// TIA Portal project "FactoryIO_Template_S7-1200_V16_V16" (V16)
// Vorlageprojekt für das Buch mit Zielsystem S7-1200

(* hardware
DEVICE "S7-1200-Station_1"  S7-1200 Station
   slot 0: "Baugruppenträger_0"  Rack  V1.0
   slot 1: "PLC_1"  CPU 1211C DC/DC/DC  6ES7 211-1AE40-0XB0  V4.1
*)

// ===== PLC "PLC_1"  CPU 1211C DC/DC/DC =====

VAR_GLOBAL   // PLC tag table "Standard-Variablentabelle"
   "EMITTER(1)" AT %A0.0 : Bool;
   "START(1)" AT %E0.0 : Bool;
   "STOP(1)" AT %E0.1 : Bool;
   "ROLLER 1" AT %Q0.1 : Bool;
   "ROLLER 2" AT %Q0.2 : Bool;
   "B LIMIT" AT %I0.3 : Bool;
   "ROLLER 4" AT %Q0.3 : Bool;
   "LIMIT 90" AT %I0.4 : Bool;
   "TURN" AT %Q0.4 : Bool;
   "ROLL +" AT %Q0.5 : Bool;
   "F LIMIT" AT %I0.2 : Bool;
   "LIMIT 0" AT %I0.5 : Bool;
   "ROLL --" AT %Q0.6 : Bool;
   "SENSOR 1" AT %I0.6 : Bool;
   "SENSOR 3" AT %I0.7 : Bool;
   "SENSOR 4" AT %I1.0 : Bool;
   "MARKER 1" AT %M0.1 : Bool;
   "MARKER 2" AT %M0.2 : Bool;
   "MARKER 3" AT %M0.3 : Bool;
   "MARKER 4" AT %M0.4 : Bool;
   "MARKER 5" AT %M0.5 : Bool;
   "MARKER 6" AT %M0.6 : Bool;
END_VAR

// folder: System blocks/Program resources

DATA_BLOCK "C1"   // DB2
{ S7_Optimized_Access := 'TRUE' }
AUTHOR : Simatic
FAMILY : IEC
NAME : CNTR
VERSION : 1.0
// stored: InstanceOfName IEC_COUNTER
"IEC_COUNTER"
BEGIN
END_DATA_BLOCK

// folder: (top level)

FUNCTION "MHJ-PLC-Lab-Function-S71200" : Void   // FC9000, SCL
{ S7_Optimized_Access := 'TRUE' }
VERSION : 0.1
   VAR_TEMP
      rdTimeReturn : Int;
      outputTime : DTL;
      SyncVal : Byte;
      forVal : Int;
      forVal_2 : Int;
      Value : Byte;
   END_VAR
   VAR CONSTANT
      CompVal : Byte := 16#34;
      Value_01 : Byte := 16#11;
      Value_01_DW : DWord := 16#A165_D992;
      Value_02_DW : DWord := 16#58BE_4401;
   END_VAR
BEGIN

   #Value:=PEEK(area := 16#82,
        dbNumber := 0,
        byteOffset := 511);
   #Value := #Value + 1;

   POKE(area := 16#82,
        dbNumber := 0,
        byteOffset := 511,
        value := #Value);

   POKE(area:=16#81,
        dbNumber:=0,
        byteOffset:=1016,
        value:=#Value_01_DW);
   POKE(area := 16#81,
        dbNumber := 0,
        byteOffset := 1020,
        value := #Value_02_DW);

   POKE(area := 16#81,
        dbNumber := 0,
        byteOffset := 511,
        value := B#16#00);

   FOR #forVal := 0 TO 120 DO
       FOR #forVal_2:=0 TO 10 DO
           #rdTimeReturn:=RD_SYS_T(#outputTime);
           #rdTimeReturn := WR_SYS_T(#outputTime);
           #rdTimeReturn := RD_SYS_T(#outputTime);
           #rdTimeReturn := WR_SYS_T(#outputTime);
       END_FOR;
       #SyncVal:= PEEK(area := 16#81,
                      dbNumber := 0,
                      byteOffset := 511);
       IF #SyncVal = #CompVal THEN
          GOTO M_1;
       END_IF;
   END_FOR;
   RETURN;

   M_1:
   POKE(area := 16#81,
        dbNumber := 0,
        byteOffset := 511,
        value := B#16#0);
END_FUNCTION

ORGANIZATION_BLOCK "Main"   // OB1, LAD, ProgramCycle
TITLE = "Main Program Sweep (Cycle)"
{ S7_Optimized_Access := 'TRUE' }
VERSION : 0.1
   VAR_INPUT
      Initial_Call : Bool;   // Initial call of this OB
      Remanence : Bool;   // =True, if remanent data are available
   END_VAR
   VAR_TEMP   // added for the SCL form of the ladder/FBD networks
      _w1 : Bool;
   END_VAR
BEGIN

REGION Network 1: Konnektierungsbaustein für PLC-Lab
   // Im Netzwerk 1 wird der Konnektierungsbaustein für PLC-Lab aufgerufen.
   // Dieser Aufruf darf nicht entfernt werden!
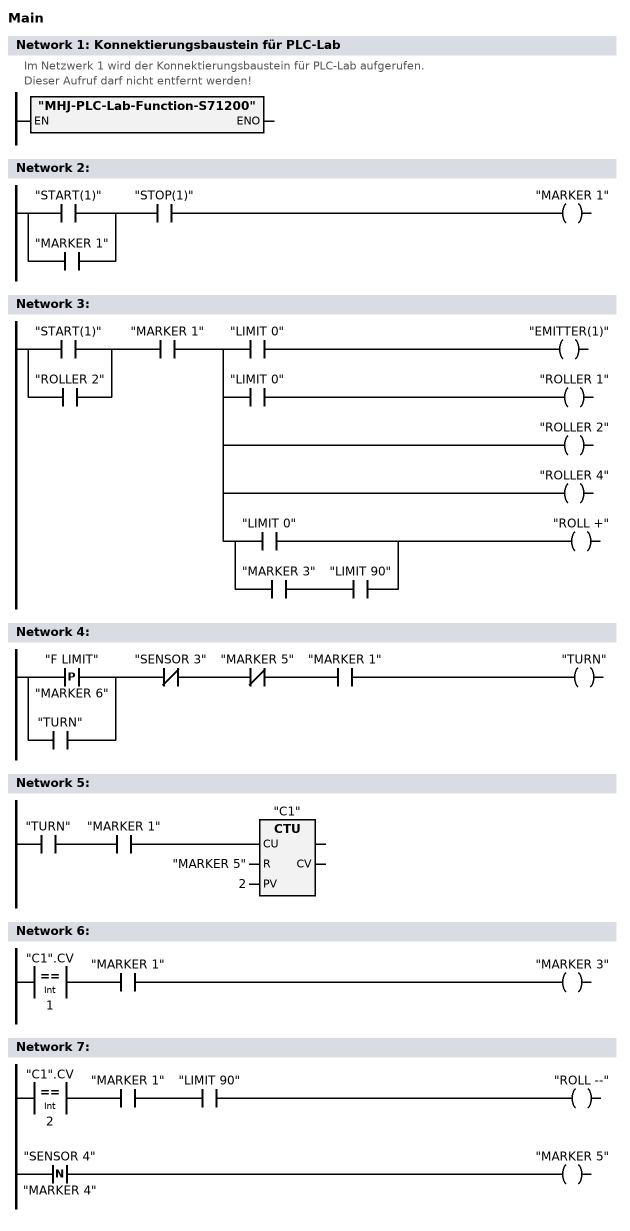
   RUNG wire#powerrail
      "MHJ-PLC-Lab-Function-S71200"()
   END_RUNG
   // the same network as SCL:
   "MHJ-PLC-Lab-Function-S71200"();
END_REGION

REGION Network 2
   RUNG wire#powerrail
      Contact( "START(1)" )
      wire#w1
      Contact( "STOP(1)" )
      Coil( "MARKER 1" )
   END_RUNG
   RUNG wire#powerrail
      Contact( "MARKER 1" )
   END_RUNG wire#w1
   // the same network as SCL:
   "MARKER 1" := ("START(1)" OR "MARKER 1") AND "STOP(1)";
END_REGION

REGION Network 3
   RUNG wire#powerrail
      Contact( "START(1)" )
      wire#w1
      Contact( "MARKER 1" )
      wire#w2
      Contact( "LIMIT 0" )
      Coil( "EMITTER(1)" )
   END_RUNG
   RUNG wire#powerrail
      Contact( "ROLLER 2" )
   END_RUNG wire#w1
   RUNG wire#w2
      Contact( "LIMIT 0" )
      Coil( "ROLLER 1" )
   END_RUNG
   RUNG wire#w2
      Coil( "ROLLER 2" )
   END_RUNG
   RUNG wire#w2
      Coil( "ROLLER 4" )
   END_RUNG
   RUNG wire#w2
      Contact( "LIMIT 0" )
      wire#w3
      Coil( "ROLL +" )
   END_RUNG
   RUNG wire#w2
      Contact( "MARKER 3" )
      Contact( "LIMIT 90" )
   END_RUNG wire#w3
   // the same network as SCL:
   #_w1 := ("START(1)" OR "ROLLER 2") AND "MARKER 1";
   "EMITTER(1)" := #_w1 AND "LIMIT 0";
   "ROLLER 1" := #_w1 AND "LIMIT 0";
   "ROLLER 2" := #_w1;
   "ROLLER 4" := #_w1;
   "ROLL +" := #_w1 AND ("LIMIT 0" OR ("MARKER 3" AND "LIMIT 90"));
END_REGION

REGION Network 4
   RUNG wire#powerrail
      P_Contact(operand := "F LIMIT", bit := "MARKER 6")
      wire#w1
      I_Contact( "SENSOR 3" )
      I_Contact( "MARKER 5" )
      Contact( "MARKER 1" )
      Coil( "TURN" )
   END_RUNG
   RUNG wire#powerrail
      Contact( "TURN" )
   END_RUNG wire#w1
   // the same network as SCL:
   #_w1 := "F LIMIT" AND NOT "MARKER 6";   // rising edge of "F LIMIT"
   "MARKER 6" := "F LIMIT";
   "TURN" := (#_w1 OR "TURN") AND NOT "SENSOR 3" AND NOT "MARKER 5" AND "MARKER 1";
END_REGION

REGION Network 5
   "C1".CTU(CU := "TURN" AND "MARKER 1", R := "MARKER 5", PV := 2);
END_REGION

REGION Network 6
   RUNG wire#powerrail
      { S7_Templates := "SrcType := Int" } EQ_Contact(in1 := "C1".CV, in2 := 1)
      Contact( "MARKER 1" )
      Coil( "MARKER 3" )
   END_RUNG
   // the same network as SCL:
   "MARKER 3" := ("C1".CV = 1) AND "MARKER 1";
END_REGION

REGION Network 7
   RUNG wire#powerrail
      { S7_Templates := "SrcType := Int" } EQ_Contact(in1 := "C1".CV, in2 := 2)
      Contact( "MARKER 1" )
      Contact( "LIMIT 90" )
      Coil( "ROLL --" )
   END_RUNG
   RUNG wire#powerrail
      N_Contact(operand := "SENSOR 4", bit := "MARKER 4")
      Coil( "MARKER 5" )
   END_RUNG
   // the same network as SCL:
   "ROLL --" := ("C1".CV = 2) AND "MARKER 1" AND "LIMIT 90";
   #_w1 := NOT "SENSOR 4" AND "MARKER 4";   // falling edge of "SENSOR 4"
   "MARKER 4" := "SENSOR 4";
   "MARKER 5" := #_w1;
END_REGION
END_ORGANIZATION_BLOCK